// TwinCAT 3 PLC project cpu
// ProgramVersion: 3.1.4024.0
// libraries:
//   Tc2_Standard, * (Beckhoff Automation GmbH)
//   Tc2_System, * (Beckhoff Automation GmbH)
//   Tc2_Utilities, * (Beckhoff Automation GmbH)
//   Tc3_IotBase, * (Beckhoff Automation GmbH)
//   Tc3_JsonXml, * (Beckhoff Automation GmbH)
//   Tc3_Module, * (Beckhoff Automation GmbH)
// project tree:
//   DUTs/ JSON_DriveList.TcDUT, JSON_Drive.TcDUT, MQTTClientStates.TcDUT, PrgStates.TcDUT
//   GVLs/ gvlMQTTConst.TcGVL
//   / MAIN.TcPOU, PlcTask.TcTTO
//   POUs/ IMQTTMsgDecoder.TcIO, MQTTClient.TcPOU, MQTTDecoder.TcPOU
// real-time tasks:
//   TASK PlcTask: cycle T#10ms, priority 20, ADS port 350

CONFIGURATION cpu
    RESOURCE PLC ON TwinCAT3
        TASK PlcTask(INTERVAL := T#10ms, PRIORITY := 20);
        PROGRAM MAIN WITH PlcTask : MAIN;
    END_RESOURCE
END_CONFIGURATION

// ---- DUTs/JSON_DriveList.TcDUT
TYPE JSON_DriveList : ARRAY[0..39] OF JSON_Drive; END_TYPE

// ---- DUTs/JSON_Drive.TcDUT
TYPE JSON_Drive :
	STRUCT
		  id 		: DINT;
		  name 		: STRING(255);
		  speed 	: LREAL;
		  torquerel : LREAL;
		  torque	: LREAL;
	END_STRUCT
END_TYPE

// ---- DUTs/MQTTClientStates.TcDUT
{attribute 'qualified_only'}
{attribute 'strict'}
TYPE MQTTClientStates :
(
	START 	:= 0,
	CONNECT := 1,
	RUN		:= 2
) DINT;
END_TYPE

// ---- DUTs/PrgStates.TcDUT
{attribute 'qualified_only'}
{attribute 'strict'}
TYPE PrgStates :
(
	START 		:= 0,
	CONNECTING 	:= 1,
	SUBSCRIBING := 2,
	RUN 		:=3
) DINT;
END_TYPE

// ---- GVLs/gvlMQTTConst.TcGVL
{attribute 'qualified_only'}
VAR_GLOBAL CONSTANT
	BUFFER_SIZE 		: DINT := 20000;
	TOPIC_SIZE			: DINT := 255;
END_VAR

// ---- POUs/IMQTTMsgDecoder.TcIO
INTERFACE IMQTTMsgDecoder

METHOD decode : BOOL
VAR_INPUT
	Topic		: REFERENCE TO STRING;
	Data		: REFERENCE TO STRING;
END_VAR
END_METHOD

END_INTERFACE

// ---- MAIN.TcPOU
PROGRAM MAIN
VAR
	decoder : MQTTDecoder;
	client : MQTTClient(Addr:='10.0.0.99', Port:=1883, MessageDecoder:=decoder);

	msg : STRING(gvlMQTTConst.BUFFER_SIZE);
	topic : STRING(gvlMQTTConst.TOPIC_SIZE) := '001/drives';
	drives : JSON_DriveList;

	N : DINT;
	
	json : FB_JsonSaxWriter;
	jsonDataType : FB_JsonReadWriteDataType;
	
	timer : TON := (PT:=T#1S);	
	state : PrgStates;
;END_VAR


timer(IN := NOT timer.Q);
client.udpate();

CASE state OF 
	PrgStates.START: 
		client.start();
		state := PrgStates.CONNECTING;
	
	PrgStates.CONNECTING:
		IF client.Connected THEN
			state := PrgStates.SUBSCRIBING;
		END_IF

	PrgStates.SUBSCRIBING:
		client.subscribe('001/call');
		state := PrgStates.RUN;

	PrgStates.RUN:
		IF timer.Q THEN
			json.ResetDocument();
			jsonDataType.AddJsonValueFromSymbol(json, 'JSON_DriveList', SIZEOF(drives), ADR(drives));
			json.CopyDocument(msg, SIZEOF(msg));
		
			client.publish(topic, ADR(msg), SIZEOF(msg));
		
			drives[0].id := N;
			N := N + 1;
		END_IF		
END_CASE

END_PROGRAM

// ---- POUs/MQTTDecoder.TcPOU
{attribute 'no_explicit_call' := 'do not call this POU directly'} 
FUNCTION_BLOCK MQTTDecoder IMPLEMENTS IMQTTMsgDecoder
VAR
	mqttData	: STRING(20000);
	mqttTopic	: STRING(1000);
END_VAR

METHOD decode : BOOL
VAR_INPUT
	Topic		: REFERENCE TO STRING;
	Data		: REFERENCE TO STRING;
END_VAR
VAR_INST
		
END_VAR

IF Topic = '001/call' THEN
	mqttData := Data;
ELSE
	mqttData := Data;	
END_IF
END_METHOD

END_FUNCTION_BLOCK

// ---- POUs/MQTTClient.TcPOU
{attribute 'no_explicit_call' := 'do not call this POU directly'} 
FUNCTION_BLOCK MQTTClient
VAR
	addr				: STRING(255);
	port				: UINT;
	msgDecoder			: IMQTTMsgDecoder;
	
	state				: MQTTClientStates;
	
	signal_connected	: BOOL;
	signal_startup		: BOOL;
	
    mqttClient  		: TC3_IOTBase.FB_IotMqttClient;
	mqttQueue			: TC3_IOTBase.FB_IotMqttMessageQueue;
	mqttMsg				: TC3_IOTBase.FB_IotMqttMessage;
	mqttBuffer			: STRING(gvlMQTTConst.BUFFER_SIZE);
	mqttTopic			: STRING(gvlMQTTConst.TOPIC_SIZE);
END_VAR

METHOD PROTECTED _maintainSignals : BOOL
signal_connected := mqttClient.bConnected;
END_METHOD

PROPERTY Connected : BOOL
GET
Connected := signal_connected;
END_GET
END_PROPERTY

METHOD FB_init : BOOL
VAR_INPUT
	bInitRetains : BOOL; // if TRUE, the retain variables are initialized (warm start / cold start)
	bInCopyCode : BOOL;  // if TRUE, the instance afterwards gets moved into the copy code (online change)
	Addr					: STRING(255);
	Port					: UINT;
	MessageDecoder			: IMQTTMsgDecoder;
END_VAR
THIS^.addr := Addr;
THIS^.port := Port;
THIS^.msgDecoder := MessageDecoder;
END_METHOD

METHOD publish : BOOL
VAR_INPUT
	Topic		: REFERENCE TO STRING;
	Data		: POINTER TO STRING;
	DataSize	: UDINT;
END_VAR

mqttClient.Publish(
	Topic,
	Data,
	LEN2(Data),
	TC3_IOTBase.TcIotMqttQos.AtLeastOnceDelivery,
	FALSE,
	FALSE
);
END_METHOD

METHOD reset : BOOL
VAR_INPUT
END_VAR
state := MQTTClientStates.START;
END_METHOD

METHOD start : BOOL
signal_startup := True;
END_METHOD

METHOD subscribe : BOOL
VAR_INPUT
	Topic : STRING(1000);
END_VAR
mqttClient.Subscribe(Topic, TC3_IoTBase.TcIotMqttQos.AtLeastOnceDelivery);
END_METHOD

METHOD udpate : BOOL

_maintainSignals();

CASE state OF
	MQTTClientStates.START:
		mqttClient.Execute(FALSE);
		IF signal_startup THEN
			signal_startup := FALSE;
			mqttClient.sHostName := addr;
			mqttClient.nHostPort := port;
			mqttClient.sTopicPrefix := '';
			mqttClient.ipMessageQueue := mqttQueue;
			state := MQTTClientStates.CONNECT;
		END_IF
		
	MQTTClientStates.CONNECT:
		mqttClient.Execute(TRUE);
		IF mqttClient.bConnected THEN
			state := MQTTClientStates.RUN;
		END_IF
	
	MQTTClientStates.RUN:
		IF NOT mqttClient.bConnected THEN
			mqttClient.Execute(FALSE);			
			state := MQTTClientStates.CONNECT;
		ELSE
			mqttClient.Execute(TRUE);
			IF msgDecoder <> 0 THEN
				IF mqttQueue.nQueuedMessages > 0 AND mqttQueue.Dequeue(mqttMsg) THEN
					mqttMsg.GetTopic(pTopic:=ADR(mqttTopic), nTopicSize:=SIZEOF(mqttTopic));
					mqttMsg.GetPayload(pPayload := ADR(mqttBuffer), nPayloadSize:=SIZEOF(mqttBuffer), bSetNullTermination := FALSE);
					msgDecoder.decode(Topic:=mqttTopic, Data:=mqttBuffer);
				END_IF
			END_IF
		END_IF
END_CASE
END_METHOD

END_FUNCTION_BLOCK
